Yaskawa INFORM job: MAIN.JBI

/JOB
//NAME MAIN
//POS
///NPOS 0,0,0,0,0,0
//INST
///DATE 2023/08/22 10:31
///ATTR SC,RW
NOP
PSTART JOB:R1_MAIN SUB1
PSTART JOB:R2_MAIN SUB2
END
